{attribute 'Tc2GvlVarNames'}
{attribute 'strict'}
TYPE e_Stato_Apprendimento :
(
	NOT_DEFINED					:= -1,  (* Apprendimendo Indefinito *)
	APPRENDIMENTO_DISABILITATO 	:= 0, 	(* Identifica che l'apprendimento NON DEVE essere eseguito *)
	APPRENDIMENTO_DA_ESEGUIRE	:= 1, 	(* Identifica che l'apprendimento DEVE essere eseguito *)
	APPRENDIMENTO_ESEGUITO		:= 2 	(* Identifica L'AVVENUTA esecuzione dell'apprendimento*)
);
END_TYPE
//  NOT_DEFINED = '-1'

(* stored: Version 1.1.0.1, ProductVersion 3.1.4024.11
   EnumerationTextList e_Stato_Apprendimento: Id {2d84f9d5-2681-4f24-945d-eae2c3c0c363} *)
